Fanuc TP program (LS listing): SHIP.LS

/PROG  SHIP
/ATTR
OWNER		= MNEDITOR;
COMMENT		= "";
PROG_SIZE	= 480;
CREATE		= DATE 22-03-26  TIME 13:24:34;
MODIFIED	= DATE 22-03-26  TIME 13:24:34;
FILE_NAME	= ;
VERSION		= 0;
LINE_COUNT	= 1;
MEMORY_SIZE	= 848;
PROTECT		= READ_WRITE;
TCD:  STACK_SIZE	= 0,
      TASK_PRIORITY	= 50,
      TIME_SLICE	= 0,
      BUSY_LAMP_OFF	= 0,
      ABORT_REQUEST	= 0,
      PAUSE_REQUEST	= 0;
DEFAULT_GROUP	= 1,*,*,*,*;
CONTROL_CODE	= 00000000 00000000;
/APPL
/APPL

AUTO_SINGULARITY_HEADER;
  ENABLE_SINGULARITY_AVOIDANCE   : TRUE;
/MN
   1:J P[1] 20% CNT100    ;
/POS
P[1]{
   GP1:
	UF : 1, UT : 1,
	J1=   168.921 deg,	J2=   -44.592 deg,	J3=   -28.000 deg,
	J4=     -.003 deg,	J5=   -43.552 deg,	J6=   183.203 deg
};
/END
